DATA_BLOCK "FB_Pointers_DB"
{ S7_Optimized_Access := 'TRUE' }
VERSION : 0.1
NON_RETAIN
"FB_Pointers"

BEGIN

END_DATA_BLOCK

